Omron CX-Programmer project NewProject (CX-Programmer 9.03)

# PLC NewPLC1: CJ1M CPU12
I/O table (CPU CJ1M-CPU12): rack 0 slot 0 CJ1W-ETN21(ETN21Mode); rack 0 slot 1 CJ1W-MAD42; rack 0 slot 2 CJ1W-ID211; rack 0 slot 3 CJ1W-OC211

## Global symbols (name address type ; comment)
0.07 BOOL  ; Start_Button
Contact _CPU007_MakeClockPulse_BCD
Start_Up_Delay _CPU003_TON_BCD

## Program NewProgram1 (cyclic task 0)
Local symbols
Annoying_Buzzer 1.07 BOOL  ; 0001.07
Comp_Flag_0 1.00 BOOL  ; 01.00
Comp_Flag_1 1.01 BOOL  ; 01.01
Comp_Flag_2 1.02 BOOL  ; 01.02
Comp_Flag_3 1.03 BOOL  ; 01.03
Comp_Flag_4 1.04 BOOL  ; 01.04
Counter C0000 BOOL  ; C0
Counter_Complete 1.06 BOOL  ; 0001.06
E_Light 1.06 BOOL  ; 0001.06
E_Stop 0.06 BOOL  ; 0000.06
Filling_0 50.00 BOOL  ; 50.00
Filling_1 50.01 BOOL  ; 50.01
Filling_2 50.02 BOOL  ; 50.02
Filling_3 50.03 BOOL  ; 50.03
Filling_4 50.04 BOOL  ; 50.04
High_Pump 1.09 BOOL  ; 0001.09
Keep_Output W0.01 BOOL  ; W00.01
Keep_Stop_Start W0.02 BOOL  ; W00.02
Low_Pump 1.08 BOOL  ; 0001.08
Low_Sensor 0.08 BOOL  ; 0000.08
Start_Relay W0.00 BOOL  ; W00.00
Start_Sensor 0.09 BOOL  ; 0000.09
Start_delay W0.15 BOOL  ; W15
Stop_Sensor 0.10 BOOL  ; 0000.10
light 1.05 BOOL  ; 0001.05

### Section Section1

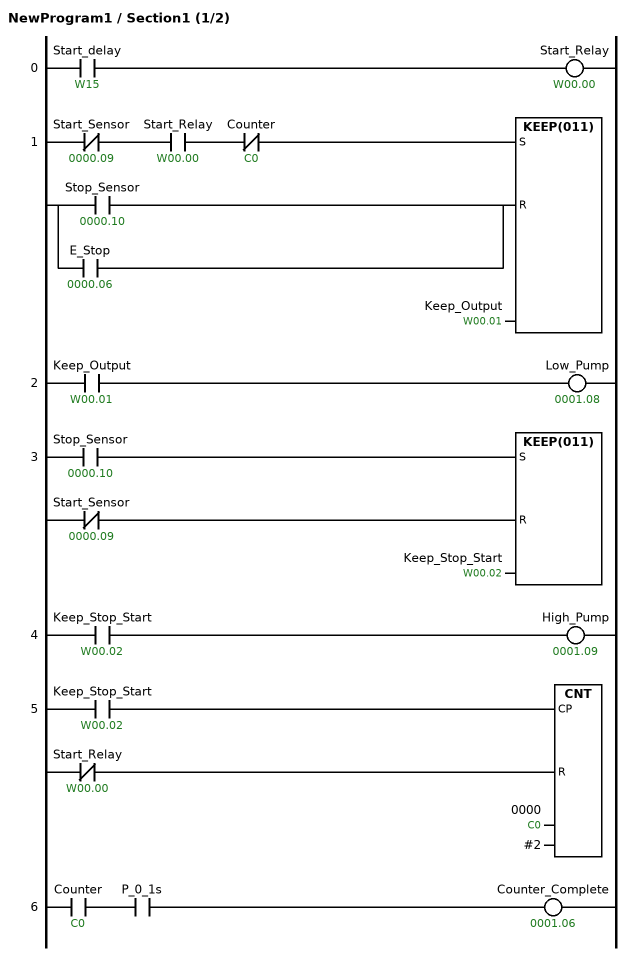
; rung 0
LD Start_delay  ; W15
OUT Start_Relay  ; W00.00
; rung 1
LDNOT Start_Sensor  ; 0000.09
AND Start_Relay  ; W00.00
ANDNOT Counter  ; C0
LD Stop_Sensor  ; 0000.10
OR E_Stop  ; 0000.06
KEEP(011) Keep_Output  ; W00.01
; rung 2
LD Keep_Output  ; W00.01
OUT Low_Pump  ; 0001.08
; rung 3
LD Stop_Sensor  ; 0000.10
LDNOT Start_Sensor  ; 0000.09
KEEP(011) Keep_Stop_Start  ; W00.02
; rung 4
LD Keep_Stop_Start  ; W00.02
OUT High_Pump  ; 0001.09
; rung 5
LD Keep_Stop_Start  ; W00.02
LDNOT Start_Relay  ; W00.00
CNT 0000 #2  ; C0
; rung 6
LD Counter  ; C0
AND P_0_1s
OUT Counter_Complete  ; 0001.06

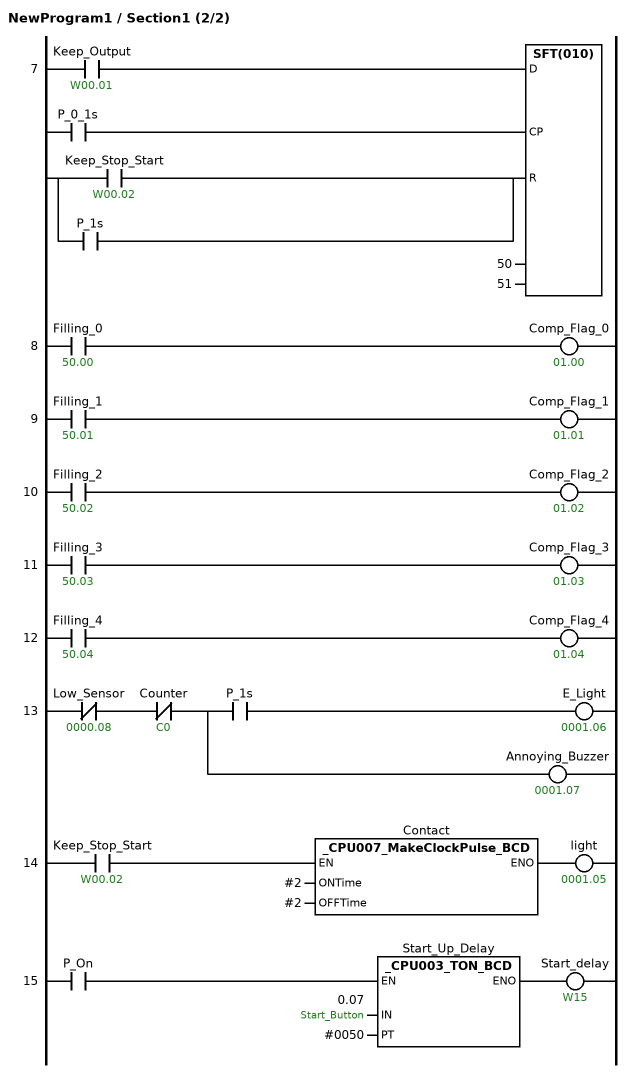
; rung 7
LD Keep_Output  ; W00.01
LD P_0_1s
LD Keep_Stop_Start  ; W00.02
OR P_1s
SFT(010) 50 51
; rung 8
LD Filling_0  ; 50.00
OUT Comp_Flag_0  ; 01.00
; rung 9
LD Filling_1  ; 50.01
OUT Comp_Flag_1  ; 01.01
; rung 10
LD Filling_2  ; 50.02
OUT Comp_Flag_2  ; 01.02
; rung 11
LD Filling_3  ; 50.03
OUT Comp_Flag_3  ; 01.03
; rung 12
LD Filling_4  ; 50.04
OUT Comp_Flag_4  ; 01.04
; rung 13
LDNOT Low_Sensor  ; 0000.08
ANDNOT Counter  ; C0
OUT TR0
AND P_1s
OUT E_Light  ; 0001.06
LD TR0
OUT Annoying_Buzzer  ; 0001.07
; rung 14
LD Keep_Stop_Start  ; W00.02
CALL Contact : _CPU007_MakeClockPulse_BCD (ONTime := #2, OFFTime := #2)
OUT light  ; 0001.05
; rung 15
LD P_On
CALL Start_Up_Delay : _CPU003_TON_BCD (IN := 0.07, PT := #0050)  ; Start_Button
OUT Start_delay  ; W15

### Section END
; rung 0
END(001)

## Function block _CPU003_TON_BCD (Omron library block, body left out)

## Function block _CPU007_MakeClockPulse_BCD (Omron library block, body left out)